{attribute 'pack_mode=1'}
TYPE BR_TrackCommand_t :
STRUCT
    enableAllSections        : BIT;
    releasePaletteAtTarget_1 : BIT;
    ApplyPaletteNumber       : BIT;
END_STRUCT
END_TYPE

(* stored: Version 1.1.0.1, ProductVersion 3.1.4024.12
   DUT BR_TrackCommand_t: Id {e97cd8b1-868e-41eb-9ffe-b3aedff7a4ec} *)
